# EPICS substitutions: mpexApp/Db/sim.substitutions
file "sim_chamber.db" {
    pattern { SYS, TTRAIN }
    { "VAC_PMI", "VAC_PMIT"  }
}
